FUNCTION_BLOCK FB_DCLINK
VAR_INPUT
	fTresholdVoltage:		REAL;
END_VAR
VAR_OUTPUT
	DC_LINK_SAFE_LEVI:		BOOL;
	DC_LINK_SAFE_PROP:		BOOL;
END_VAR
VAR
END_VAR

//DC-LINK LEVI
IF GVL_LEVI.drive_voltage_EMS1 < fTresholdVoltage
AND GVL_LEVI.drive_voltage_EMS2 < fTresholdVoltage 
AND GVL_LEVI.drive_voltage_EMS3 < fTresholdVoltage
AND GVL_LEVI.drive_voltage_EMS4 < fTresholdVoltage
AND GVL_LEVI.drive_voltage_HEMS1 < fTresholdVoltage
AND GVL_LEVI.drive_voltage_HEMS2 < fTresholdVoltage
AND GVL_LEVI.drive_voltage_HEMS3 < fTresholdVoltage
AND GVL_LEVI.drive_voltage_HEMS4 < fTresholdVoltage
AND GVL_LEVI.drive_voltage_HEMS5 < fTresholdVoltage
AND GVL_LEVI.drive_voltage_HEMS6 < fTresholdVoltage
AND GVL_LEVI.drive_voltage_HEMS7 < fTresholdVoltage
AND GVL_LEVI.drive_voltage_HEMS8 < fTresholdVoltage THEN

	DC_LINK_SAFE_LEVI := TRUE;
	
END_IF


//DC-LINK PROP
IF GVL_Prop.drive_voltages1 < 60.0 
AND GVL_Prop.drive_voltages2 < 60.0
AND GVL_Prop.drive_voltages3 < 60.0
AND GVL_Prop.drive_voltages4 < 60.0 THEN
	
	DC_LINK_SAFE_PROP := TRUE;

END_IF

END_FUNCTION_BLOCK

(* stored: Version 1.1.0.1
   POU FB_DCLINK: Id {0fb4be52-4f9e-4920-af05-61e385489610}, SpecialFunc None *)
